{attribute addProperty BoxType "IODEVICETYPE_ETHERCATPROT"}
{attribute addProperty Id "Beckhoff_EQ1xxxBeckhoff_EQ1xxx_788CB99A62478Beckhoff_EQ2xxxBeckhoff_EQ2xxx_1D920FDF1976247Beckhoff_EQ3xxxBeckhoff_EQ3xxx_C3FDE44A3656457SyncUnitsSyncUnits_3FA29F3C21627InputsInputs_C75D3FEC1280160OutputsOutputs_47D1E803848106InfoDataInfoData_45F98C5022428"}
{attribute addProperty CRC "98099514"}
{attribute addProperty SizeInBites "8824"}
{attribute addProperty SizeInBytes "1103"}
TYPE EtherCAT_Master_EQxxxx_05D8E13A :
STRUCT
	{attribute addProperty Name "Beckhoff_EQ1xxx"}
	Beckhoff_EQ1xxx : Beckhoff_EQ1xxx_788CB99A;
	{attribute addProperty Name "Beckhoff_EQ2xxx"}
	Beckhoff_EQ2xxx : Beckhoff_EQ2xxx_1D920FDF;
	{attribute addProperty Name "Beckhoff_EQ3xxx"}
	Beckhoff_EQ3xxx : Beckhoff_EQ3xxx_C3FDE44A;
	{attribute addProperty Name "SyncUnits"}
	SyncUnits : SyncUnits_3FA29F3C;
	{attribute addProperty Name "Inputs"}
	Inputs : Inputs_C75D3FEC;
	{attribute addProperty Name "Outputs"}
	Outputs : Outputs_47D1E803;
	{attribute addProperty Name "InfoData"}
	InfoData : InfoData_45F98C50;
END_STRUCT
END_TYPE

(* stored: Version 1.2.0.0, ProductVersion 3.1.4024.9
   DUT EtherCAT_Master_EQxxxx_05D8E13A: Id {b5c4827a-192f-4465-a68a-6d7e9b81e947} *)
